(* IEC 61131-3 sources: plc/, 3 files *)

(* ---- union64-converter.st ---- *)
//Can be used e.g. to split a REAL into BYTE or WORD.
//Example(s):
//- WORD <-> BYTE:	unX64.aw[0] <-> unX64.ab[0..1]
//- REAL <-> WORD:	unX64.ar[0] <-> unX64.aw[0..1]
//- REAL <-> WORD <-> BYTE:	unX64.ar[0] <-> unX64.aw[0..1] <-> unX64.ab[0..3]
/////////////////////////////////////////////////////////////////////////////////////////////////
///e.g. "2x WORD <-> REAL"///////////////////////////////////////////////////////////////////////
/////////////////////////////////////////////////////////////////////////////////////////////////
TYPE unX64 :
UNION
	lw:	LWORD;			// 1x 64Bit
	adw:	ARRAY[0..1] OF DWORD;	// 2x 32Bit
	aw:	ARRAY[0..3] OF WORD;	// 4x 16Bit
	ab:	ARRAY[0..7] OF BYTE;	// 8x  8bit

	uli:	ULINT;			// 1x 64Bit unsigned INT
	audi:	ARRAY[0..1] OF UDINT;	// 2x 32Bit unsigned INT
	aui:	ARRAY[0..3] OF UINT;	// 4x 16Bit unsigned INT
	ausi:	ARRAY[0..7] OF USINT;	// 8x  8bit unsigned INT

	li:	LINT;			// 1x 64Bit signed INT
	adi:	ARRAY[0..1] OF DINT;	// 2x 32Bit signed INT
	ai:	ARRAY[0..3] OF INT;	// 4x 16Bit signed INT
	asi:	ARRAY[0..7] OF SINT;	// 8x  8bit signed INT

	lr:	LREAL;			// 1x 64Bit REAL
	ar:	ARRAY[0..1] OF REAL;	// 2x 32Bit REAL
END_UNION
END_TYPE
/////////////////////////////////////////////////////////////////////////////////////////////////
/////////////////////////////////////////////////////////////////////////////////////////////////
VAR
	awData:	ARRAY [0..1] OF WORD;
	rVar:	REAL;
END_VAR

VAR_TEMP
	_unX64:	unX64;			// Type converter;
END_VAR
/////////////////////////////////////////////////////////////////////////////////////////////////
/////////////////////////////////////////////////////////////////////////////////////////////////
// rVar
_unX64.aw[0]	:= awData[0];
_unX64.aw[1]	:= awData[1];
rVar 		:= _unX64.ar[0];
/////////////////////////////////////////////////////////////////////////////////////////////////
/////////////////////////////////////////////////////////////////////////////////////////////////

(* ---- example-folding-issue.st ---- *)
// This file demonstrates the code folding display issue
// When you collapse the code between comments, the display is malformed

// parent instuction
	// step 1
	// step 2
	// step 3

	// step 4
	// step 5
// end of parent instruction

// Another example with actual PLC code
// Initialize system variables
	VAR
		xSystemReady: BOOL := FALSE;
		iCounter: INT := 0;
		rTemperature: REAL := 0.0;
	END_VAR
// End initialization

// Main control loop
	IF xSystemReady THEN
		iCounter := iCounter + 1;
		// Process temperature reading
		IF rTemperature > 100.0 THEN
			// Emergency shutdown
			xSystemReady := FALSE;
		END_IF;
	END_IF;
// End main control loop

(* ---- xPulse-every-200ms.st ---- *)
VAR
  tTonPulse: TON;
  xPulseOneCycle: BOOL;
END_VAR

tTonPulse(IN:= TRUE, PT:= T#200ms);
IF tTonPulse.Q THEN
    tTonPulse(IN:= FALSE);
    xPulseOneCycle := TRUE;
END_IF;

IF xPulseOneCycle THEN
    // Aquí puedes realizar las acciones que deseas mientras el xPulseOneCycle esté activo
    // Por ejemplo, encender una salida
    xPulseOneCycle := FALSE;
END_IF;
